// TwinCAT 3 PLC project PLC_HMI
// ProgramVersion: 3.1.4024.0
// libraries:
//   CmpBitmapPool, * (System)
//   Tc2_Standard, * (Beckhoff Automation GmbH)
//   Tc2_System, * (Beckhoff Automation GmbH)
//   Tc2_Utilities, * (Beckhoff Automation GmbH)
//   Tc3_Module, * (Beckhoff Automation GmbH)
//   VisuDialogs, * (System)
// project tree:
//   / GlobalTextList.TcGTLO, PlcTask.TcTTO, VisualizationManager.TcVMO (not stored), VISU_TASK.TcTTO
//   GVLs/ GVL.TcGVL
//   POUs/ FB_UpdateTimeStamp.TcPOU, MAIN.TcPOU, OP_BTN.TcPOU, SetBit.TcPOU
//   VISUs/ CONFIRMATION.TcVIS, FOOTER.TcVIS, PAGE_SYSTEM.TcVIS, PAGE_RUN.TcVIS, ImagePool.TcIPO (not stored), PAGE_HOME.TcVIS, PAGE_CONTROL.TcVIS

CONFIGURATION PLC_HMI
    RESOURCE PLC ON TwinCAT3
        TASK PlcTask(INTERVAL := T#10ms, PRIORITY := 20);
        TASK VISU_TASK(INTERVAL := T#200000us, PRIORITY := 30);
        PROGRAM MAIN WITH PlcTask : MAIN;
        PROGRAM VisuElems_Visu_Prg WITH VISU_TASK : VisuElems.Visu_Prg;
    END_RESOURCE
END_CONFIGURATION

// ---- GVLs/GVL.TcGVL
{attribute 'qualified_only'}
VAR_GLOBAL
	TableRecord		: ARRAY [1..5,1..7] OF STRING;
	TODAY			: WORD;
	YESTERDAY		: WORD;
	LASTMONTH		: UINT;
	LASTYEAR		: UINT;
	
	DailyCnt_FG1	: INT;
	DailyCnt_FG2	: INT;
	DailyCnt_FG3	: INT;
	DailyCnt_FG4	: INT;
	MonthCnt		: UINT;
	YearCnt			: UINT;
END_VAR

// ---- POUs/MAIN.TcPOU
PROGRAM MAIN
VAR
	fb_TimeStamp : FB_UpdateTimeStamp ();
END_VAR

// Open PLC HMI view here C:\TwinCAT\3.1\Components\Plc\Tc3PlcHmi
// Open PLC HMI web view with this link   http://127.0.0.1/Tc3PlcHmiWeb/Port_851/Visu/webvisu.htm


fb_TimeStamp();
OP_BTN();

END_PROGRAM

// ---- POUs/FB_UpdateTimeStamp.TcPOU
FUNCTION_BLOCK FB_UpdateTimeStamp
VAR_INPUT
END_VAR
VAR_OUTPUT
	FullSystemTime	: STRING;
	SystemYear		: STRING;
	SystemDate		: STRING;
	SystemTime		: STRING;
	SystemHour		: STRING;
	timeValid		: BOOL;
	day 	: ARRAY [1..7] OF BOOL;
END_VAR
VAR
	fb_LocalTime	: FB_LocalSystemTime;
	dayNum			: UINT;
	today 			: STRING;
END_VAR

//  --------------------------------------------------------------- Initialize
	fb_LocalTime(
			sNetID:= , 
			bEnable:= TRUE , 
			dwCycle:= 1, 
			dwOpt:= , 
			tTimeout:= ,
			bValid=> timeValid, 
			systemTime=> , 
			tzID=> );
			
//  --------------------------------------------------------------- Set system time	
	IF fb_localTime.bValid THEN
		FullSystemTime 	:= SYSTEMTIME_TO_STRING(fb_LocalTime.systemTime);
		
		SystemYear		:= WORD_TO_STRING(fb_LocalTime.systemTime.wYear);
		SystemDate		:= WORD_TO_STRING(fb_LocalTime.systemTime.wYear);
		SystemDate		:= CONCAT(SystemDate, '.');
		SystemDate		:= CONCAT(SystemDate, WORD_TO_STRING(fb_LocalTime.systemTime.wMonth));
		SystemDate		:= CONCAT(SystemDate, '.');
		SystemDate		:= CONCAT(SystemDate, WORD_TO_STRING(fb_LocalTime.systemTime.wDay));
		
		SystemTime		:= WORD_TO_STRING(fb_LocalTime.systemTime.wHour);
		SystemTime		:= CONCAT(SystemTime, ':');
		SystemTime		:= CONCAT(SystemTime, WORD_TO_STRING(fb_LocalTime.systemTime.wMinute));
		SystemTime		:= CONCAT(SystemTime, ':');
		SystemTime		:= CONCAT(SystemTime, WORD_TO_STRING(fb_LocalTime.systemTime.wSecond));
		
		SystemHour		:= WORD_TO_STRING(fb_LocalTime.systemTime.wHour);
	
		dayNum := WORD_TO_UINT(fb_localTime.systemTime.wDayOfWeek);
		GVL.TODAY := fb_localTime.systemTime.wDay;
		IF dayNum = 0 THEN
			dayNum :=1;
		END_IF
		
		GVL.TableRecord [1,dayNum] := CONCAT (WORD_TO_STRING(fb_LocalTime.systemTime.wDay),'-');
		GVL.TableRecord [1,dayNum] := CONCAT (GVL.TableRecord [1,dayNum],WORD_TO_STRING(fb_LocalTime.systemTime.wMonth));
		GVL.TableRecord [1,dayNum] := CONCAT (GVL.TableRecord [1,dayNum],'-');
		GVL.TableRecord [1,dayNum] := CONCAT (GVL.TableRecord [1,dayNum],WORD_TO_STRING(fb_LocalTime.systemTime.wYear));
		
		CASE dayNum OF
			1:
				today := 'Monday';
				day[1] := FALSE;
				day[2] := day[3] := day[4] := day[5] := day[6] := day[7] := TRUE;
			2:
				today := 'Tuesday';
				day[2] := FALSE;
				day[1] := day[3] := day[4] := day[5] := day[6] := day[7] := TRUE;
			3:
				today := 'Wednesday';
				day[3] := FALSE;
				day[1] := day[2] := day[4] := day[5] := day[6] := day[7] := TRUE;
			4:
				today := 'Thursday';
				day[4] := FALSE;
				day[1] := day[2] := day[3] := day[5] := day[6] := day[7] := TRUE;
			5:
				today := 'Friday';
				day[5] := FALSE;
				day[1] := day[2] := day[3] := day[4] := day[6] := day[7] := TRUE;
			6:
				today := 'Saturday';
				day[6] := FALSE;
				day[1] := day[2] := day[3] := day[4] := day[5] := day[7] := TRUE;
			7:
				today := 'Sunday';
				day[7] := FALSE;
				day[1] := day[2] := day[3] := day[4] := day[5] := day[6] := TRUE;
			END_CASE

	//  --------------------------------------------------------------- TABLE logging
		IF GVL.TODAY <> GVL.YESTERDAY THEN
			GVL.YESTERDAY := GVL.TODAY;
			GVL.DailyCnt_FG1 := GVL.DailyCnt_FG2 := GVL.DailyCnt_FG3 := GVL.DailyCnt_FG4 := 0;
		END_IF		
		IF GVL.LASTMONTH <> fb_LocalTime.systemTime.wMonth THEN
			GVL.LASTMONTH := fb_LocalTime.systemTime.wMonth;
			GVL.MonthCnt  := GVL.MonthCnt + 1;
		END_IF	
		IF GVL.LASTYEAR <> fb_LocalTime.systemTime.wYear THEN
			GVL.LASTYEAR := fb_LocalTime.systemTime.wYear;
			GVL.YearCnt  := GVL.YearCnt + 1;
		END_IF
		
		GVL.TableRecord [2,dayNum] := INT_TO_STRING(GVL.DailyCnt_FG1);
		GVL.TableRecord [3,dayNum] := INT_TO_STRING(GVL.DailyCnt_FG2);
		GVL.TableRecord [4,dayNum] := INT_TO_STRING(GVL.DailyCnt_FG3);
		GVL.TableRecord [5,dayNum] := INT_TO_STRING(GVL.DailyCnt_FG4);
		
	END_IF

END_FUNCTION_BLOCK

// ---- POUs/OP_BTN.TcPOU
PROGRAM OP_BTN
VAR
	Start_btn	: BOOL;
	Start_lamp	: BOOL;
	Reset_btn	: BOOL;
	Reset_lamp	: BOOL;
	Estop_btn	: BOOL;
	Estop_lamp	: BOOL;
END_VAR

// Lamp Operation 

Start_lamp := Start_btn AND NOT Reset_btn AND NOT Estop_btn;

Estop_lamp := Estop_btn AND NOT Reset_btn;


// Lamp Reset
IF Reset_btn THEN
	Start_btn := Estop_btn := FALSE;
	Reset_lamp := TRUE;
END_IF

IF Estop_btn THEN
	Start_btn := Reset_btn := FALSE;
	Reset_lamp := FALSE;
END_IF

END_PROGRAM

// ---- POUs/SetBit.TcPOU
FUNCTION SetBit : DWORD
VAR_INPUT
	dPLC_OUT	: DWORD;
	iBitNum		: USINT;
	bstate		: BOOL;
END_VAR
VAR
	bCheckBit	: BOOL;
END_VAR


bCheckBit := DWORD_TO_BOOL(SHR(dPLC_OUT,iBitNum)AND 1);

IF bstate THEN
	dPLC_OUT := SHL(1,iBitNum) OR dPLC_OUT;
ELSE
	IF bCheckbit THEN
		IF dPLC_OUT > 0 THEN
			dPLC_OUT := dPLC_OUT - LREAL_TO_DWORD(EXPT(2,iBitNum));
		END_IF
	END_IF
END_IF

SetBit := dPLC_OUT;

END_FUNCTION

// ---- GlobalTextList.TcGTLO
TEXTLIST GlobalTextList
  82 = '%s'
  217 = 'A'
  902 = 'Admin'
  132 = 'ADMIN'
  997 = 'Are you Sure ?'
  773 = 'B'
  996 = 'C'
  180 = 'Calibration'
  3105 = 'Connect   Laser'
  1339 = 'Connect Scanner'
  395 = 'Control'
  313 = 'CONTROL PAGE'
  596 = 'D'
  815 = 'Date'
  934 = 'Emergency Stop'
  153 = 'FG-1'
  767 = 'FG-2'
  89 = 'FG-3'
  417 = 'FG-4'
  133 = 'Home'
  266 = 'HOME PAGE'
  186 = 'Login'
  47 = 'LOGIN'
  735 = 'Logout'
  992 = 'LOGOUT'
  2441 = 'Mute\nBuzzer'
  532 = 'No'
  472 = 'None'
  30 = 'Operator'
  391 = 'OPERATOR'
  92 = 'Reset Button'
  885 = 'Run'
  192 = 'RUN PAGE'
  899 = 'Selected model'
  941 = 'Start Button'
  88 = 'System'
  451 = 'SYSTEM PAGE'
  608 = 'WARNING'
  412 = 'Yes'
END_TEXTLIST

// ---- VISUs/CONFIRMATION.TcVIS
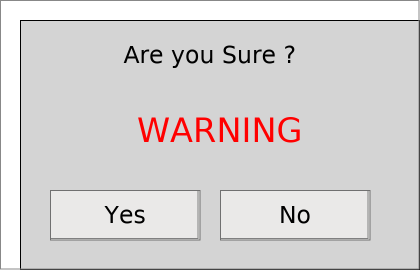
VISUALIZATION CONFIRMATION  // 420x270
VAR_IN_OUT
	result : STRING;
END_VAR
    Rectangle (20,20 400x250)
    Button (50,190 150x50), "Yes"
        toggle OP_BTN.Start_btn
        OnMouseClick: CloseDialog Dialog=CONFIRMATION, Result=Yes, NumpadKeypadSet=True
    Label (85,30 250x50), "Are you Sure ?"
    Button (220,190 150x50), "No"
        OnMouseClick: CloseDialog Dialog=CONFIRMATION, Result=No, NumpadKeypadSet=True
    Textfield (20,100 400x60), "WARNING"
END_VISUALIZATION

// ---- VISUs/FOOTER.TcVIS
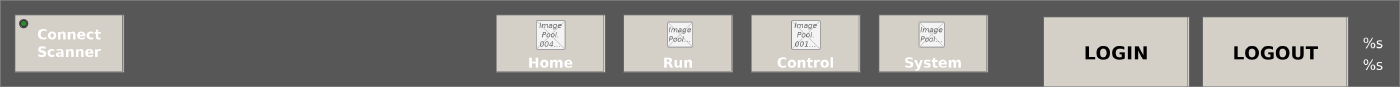
VISUALIZATION FOOTER  // 1920x120
    Textfield (1700,70 200x40), "%s", text variable: MAIN.fb_TimeStamp.SystemDate
    Textfield (1700,40 200x40), "%s", text variable: MAIN.fb_TimeStamp.SystemTime
    Group (855,20 150x80)
        OnMouseClick: change screen: PAGE_RUN
        Button (0,0 150x80), "Run"
        Image (60,10 35x35), image: ImagePool.003-play-button-arrowhead
    Group (1030,20 150x80)
        OnMouseClick: change screen: PAGE_CONTROL
        Button (0,0 150x80), "Control"
        Image (55,8 40x40), image: ImagePool.001-gear
    Group (680,20 150x80)
        OnMouseClick: change screen: PAGE_HOME
        Button (0,0 150x80), "Home"
        Image (55,8 40x40), image: ImagePool.004-home
    Group (1205,20 150x80)
        OnMouseClick: change screen: PAGE_SYSTEM
        Button (0,0 150x80), "System"
        Image (55,10 35x35), image: ImagePool.002-folder
    Button (20,20 150x80), "Connect Scanner"
    Lamp1 (25,25 15x15), style: Lamp-Lamp1-Green
    Group (1431,23 293x60)
        Button (218,0 200x100), "LOGOUT"
            OnMouseClick: VisuUserMgmt Type=Logout
        Button (0,0 200x100), "LOGIN"
            OnMouseClick: VisuUserMgmt Type=Login
END_VISUALIZATION

// ---- VISUs/PAGE_SYSTEM.TcVIS
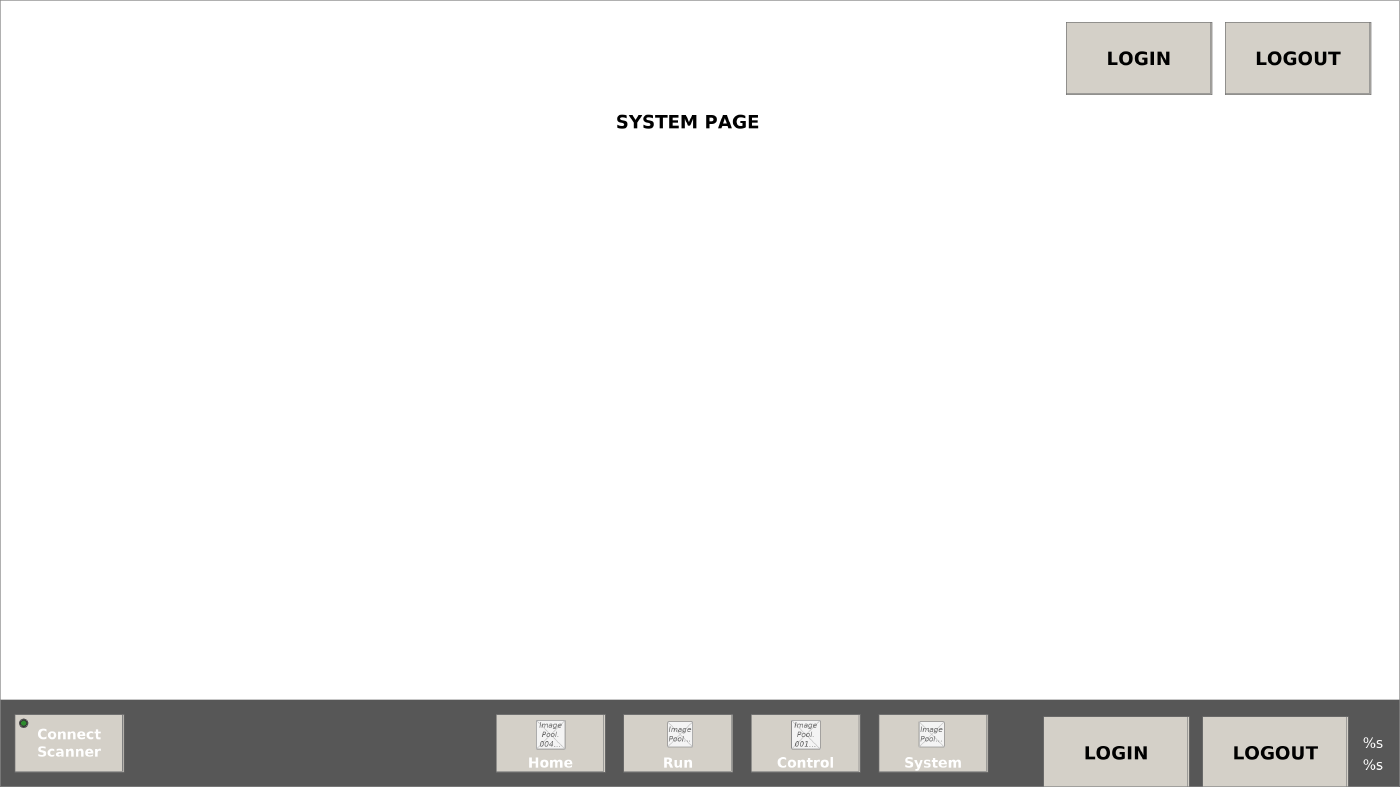
VISUALIZATION PAGE_SYSTEM  // 1920x1080, background image ImagePool.Grey_Gradient
    Button (1462,30 200x100), "LOGIN"
        OnMouseClick: VisuUserMgmt Type=Login
    Button (1680,30 200x100), "LOGOUT"
        OnMouseClick: VisuUserMgmt Type=Logout
    Frame (0,960 1920x120)
        shows FOOTER()
    Label (708,109 470x116), "SYSTEM PAGE"
END_VISUALIZATION

// ---- VISUs/PAGE_RUN.TcVIS
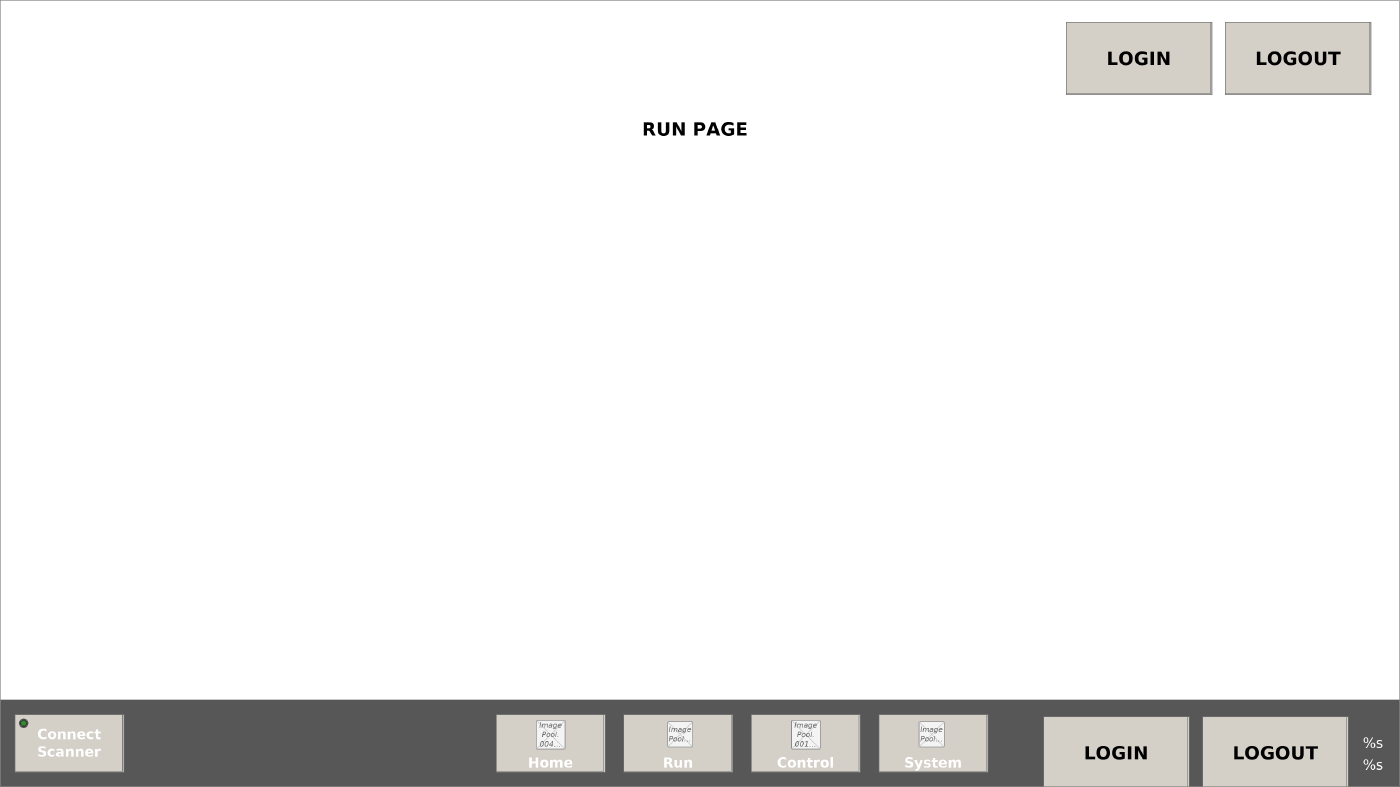
VISUALIZATION PAGE_RUN  // 1920x1080, background image ImagePool.Grey_Gradient
    Button (1462,30 200x100), "LOGIN"
        OnMouseClick: VisuUserMgmt Type=Login
    Button (1680,30 200x100), "LOGOUT"
        OnMouseClick: VisuUserMgmt Type=Logout
    Frame (0,960 1920x120)
        shows FOOTER()
    Label (718,119 470x116), "RUN PAGE"
END_VISUALIZATION

// ---- VISUs/PAGE_HOME.TcVIS
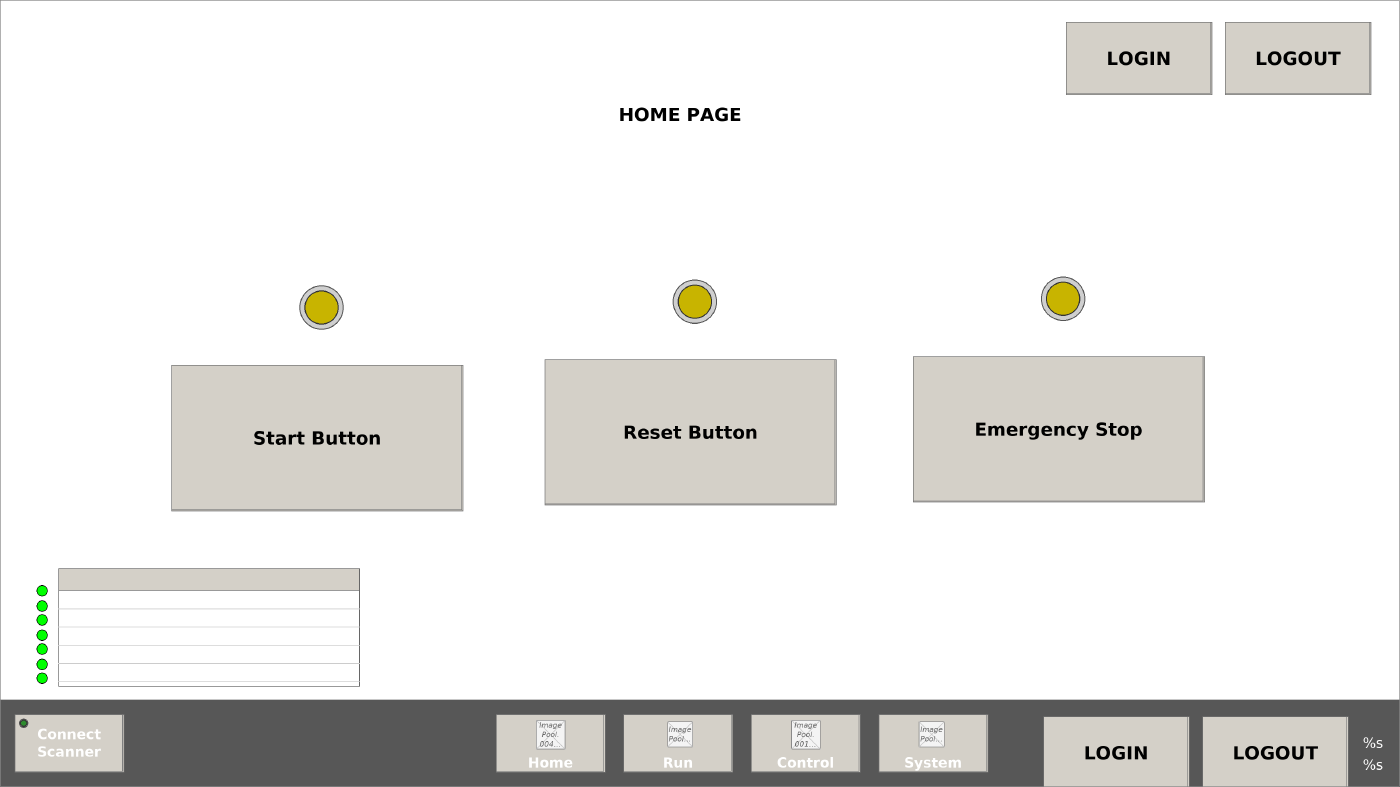
VISUALIZATION PAGE_HOME  // 1920x1080, background image ImagePool.Grey_Gradient
    Button (235,501 400x200), "Start Button"
        OnMouseClick: OpenDialog Dialog=CONFIRMATION, OpenModal=True, OpenCentered=True
    Lamp1 (406,387 70x70), variable: OP_BTN.Start_lamp, style: Lamp-Lamp1-Yellow
    Button (747,493 400x200), "Reset Button"
        tap OP_BTN.Reset_btn
    Lamp1 (918,379 70x70), variable: OP_BTN.Reset_lamp, style: Lamp-Lamp1-Yellow
    Button (1252,489 400x200), "Emergency Stop"
        toggle OP_BTN.Estop_btn
    Lamp1 (1423,375 70x70), variable: OP_BTN.Estop_lamp, style: Lamp-Lamp1-Yellow
    Button (1462,30 200x100), "LOGIN"
        OnMouseClick: VisuUserMgmt Type=Login
    Button (1680,30 200x100), "LOGOUT"
        OnMouseClick: VisuUserMgmt Type=Logout
    Frame (0,960 1920x120)
        shows FOOTER()
    Label (698,99 470x116), "HOME PAGE"
    Table (80,780 413x162), data array: GVL.TableRecord
        p3854506369: GVL.TableRecord[1,INDEX]
        p1892666644: GVL.TableRecord[2,INDEX]
        p338671338: GVL.TableRecord[3,INDEX]
        p2170511999: GVL.TableRecord[4,INDEX]
        p3723444502: GVL.TableRecord[5,INDEX]
        p2232123230: Date
        p511219082: FG-1
        p1755163831: FG-2
        p4092479075: FG-3
        p2237128397: FG-4
    Ellipse (50,803 15x15), invisible if: MAIN.fb_TimeStamp.day[1]
    Ellipse (50,824 15x15), invisible if: MAIN.fb_TimeStamp.day[2]
    Ellipse (50,843 15x15), invisible if: MAIN.fb_TimeStamp.day[3]
    Ellipse (50,864 15x15), invisible if: MAIN.fb_TimeStamp.day[4]
    Ellipse (50,883 15x15), invisible if: MAIN.fb_TimeStamp.day[5]
    Ellipse (50,904 15x15), invisible if: MAIN.fb_TimeStamp.day[6]
    Ellipse (50,923 15x15), invisible if: MAIN.fb_TimeStamp.day[7]
END_VISUALIZATION

// ---- VISUs/PAGE_CONTROL.TcVIS
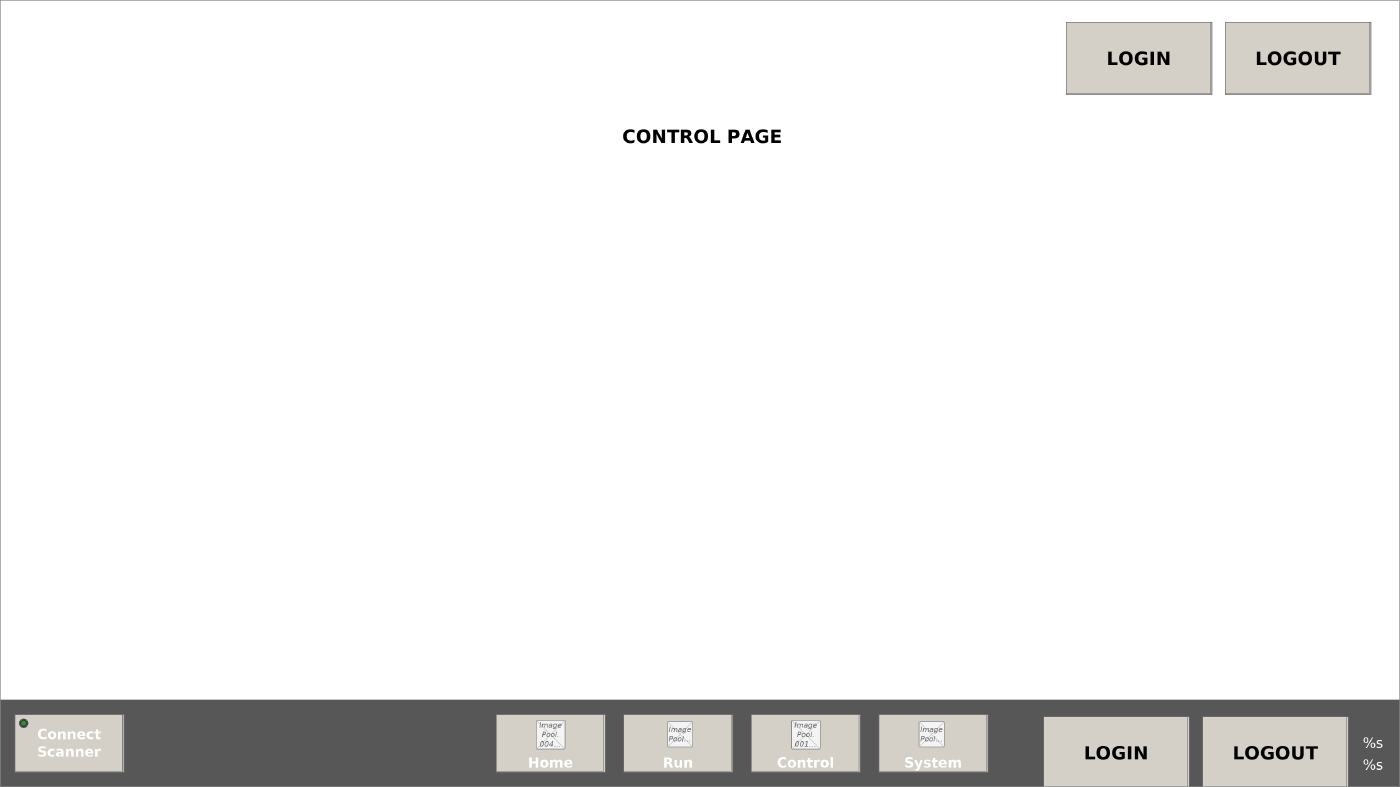
VISUALIZATION PAGE_CONTROL  // 1920x1080, background image ImagePool.Grey_Gradient
    Button (1462,30 200x100), "LOGIN"
        OnMouseClick: VisuUserMgmt Type=Login
    Button (1680,30 200x100), "LOGOUT"
        OnMouseClick: VisuUserMgmt Type=Logout
    Frame (0,960 1920x120)
        shows FOOTER()
    Label (728,129 470x116), "CONTROL PAGE"
END_VISUALIZATION
